// TwinCAT 3 PLC project MainPlc
// ProgramVersion: 3.1.4026.24
// libraries:
//   Tc2_MC2, * (Beckhoff Automation GmbH)
//   Tc2_Standard, * (Beckhoff Automation GmbH)
//   Tc2_System, * (Beckhoff Automation GmbH)
// project tree:
//   DUTs/ ST_AxisData.TcDUT (not stored)
//   GVLs/ GVL_Axis.TcGVL (not stored), GVL_CONSTANT.TcGVL, GVL_PY.TcGVL (not stored)
//   / PlcTask.TcTTO
//   POUs/Axis/ FB_AxisCtrl.TcPOU (not stored), PRG_Enable.TcPOU (not stored), PRG_SineWave.TcPOU (not stored), PRG_Square.TcPOU (not stored)
//   POUs/ MAIN.TcPOU (not stored)
// real-time tasks:
//   TASK PlcTask: cycle T#1ms, priority 20, ADS port 350
// motion (NC):
//   TASK NC-Task 1 SAF: cycle T#1ms, priority 4, ADS port 501
//   TASK NC-Task 1 SVB: cycle T#1ms, priority 8, ADS port 511
//   AXIS Axis 1 (id 1)
//     OtherSettings: AllowMotionCmdToSlave=true
//     encoder EncType=1
//       TimeComp: TimeCompMode=1, EncDelayCycles=4
//     drive DrvType=5
//       Analog: TorqueSetpointScale=10, ScaleFactorActTorque=0.1
//       TimeComp: TimeCompMode=1, TaskDelayCycles=1
//     controller CtrType=1
//       CtrPara: PriorControlFactor=1
//         Observer: BandWidth=20
//   AXIS Axis 2 (id 2)
//     OtherSettings: AllowMotionCmdToSlave=true
//     encoder EncType=1
//     drive DrvType=5
//       Analog: TorqueSetpointScale=10, ScaleFactorActTorque=0.1
//       TimeComp: TaskDelayCycles=1
//     controller CtrType=1
//       CtrPara: PriorControlFactor=1
//         Observer: BandWidth=20
//   AXIS Axis 3 (id 3)
//     OtherSettings: AllowMotionCmdToSlave=true
//     encoder EncType=1
//     drive DrvType=5
//       Analog: TorqueSetpointScale=10, ScaleFactorActTorque=0.1
//       TimeComp: TaskDelayCycles=1
//     controller CtrType=1
//       CtrPara: PriorControlFactor=1
//         Observer: BandWidth=20
//   AXIS Axis 4 (id 4)
//     OtherSettings: AllowMotionCmdToSlave=true
//     encoder EncType=1
//     drive DrvType=5
//       Analog: TorqueSetpointScale=10, ScaleFactorActTorque=0.1
//       TimeComp: TaskDelayCycles=1
//     controller CtrType=1
//       CtrPara: PriorControlFactor=1
//         Observer: BandWidth=20
//   AXIS Axis 5 (id 5)
//     OtherSettings: AllowMotionCmdToSlave=true
//     encoder EncType=1
//     drive DrvType=5
//       Analog: TorqueSetpointScale=10, ScaleFactorActTorque=0.1
//       TimeComp: TaskDelayCycles=1
//     controller CtrType=1
//       CtrPara: PriorControlFactor=1
//         Observer: BandWidth=20
//   AXIS Axis 6 (id 6)
//     OtherSettings: AllowMotionCmdToSlave=true
//     encoder EncType=1
//     drive DrvType=5
//       Analog: TorqueSetpointScale=10, ScaleFactorActTorque=0.1
//       TimeComp: TaskDelayCycles=1
//     controller CtrType=1
//       CtrPara: PriorControlFactor=1
//         Observer: BandWidth=20
//   AXIS Axis 7 (id 7)
//     OtherSettings: AllowMotionCmdToSlave=true
//     encoder EncType=1
//     drive DrvType=5
//       Analog: TorqueSetpointScale=10, ScaleFactorActTorque=0.1
//       TimeComp: TaskDelayCycles=1
//     controller CtrType=1
//       CtrPara: PriorControlFactor=1
//         Observer: BandWidth=20
//   AXIS Axis 8 (id 8)
//     OtherSettings: AllowMotionCmdToSlave=true
//     encoder EncType=1
//     drive DrvType=5
//       Analog: TorqueSetpointScale=10, ScaleFactorActTorque=0.1
//       TimeComp: TaskDelayCycles=1
//     controller CtrType=1
//       CtrPara: PriorControlFactor=1
//         Observer: BandWidth=20
//   AXIS Axis 9 (id 9)
//     OtherSettings: AllowMotionCmdToSlave=true
//     encoder EncType=1
//     drive DrvType=5
//       Analog: TorqueSetpointScale=10, ScaleFactorActTorque=0.1
//       TimeComp: TaskDelayCycles=1
//     controller CtrType=1
//       CtrPara: PriorControlFactor=1
//         Observer: BandWidth=20
//   AXIS Axis 10 (id 10)
//     OtherSettings: AllowMotionCmdToSlave=true
//     encoder EncType=1
//     drive DrvType=5
//       Analog: TorqueSetpointScale=10, ScaleFactorActTorque=0.1
//       TimeComp: TaskDelayCycles=1
//     controller CtrType=1
//       CtrPara: PriorControlFactor=1
//         Observer: BandWidth=20
//   AXIS Axis 11 (id 11)
//     OtherSettings: AllowMotionCmdToSlave=true
//     encoder EncType=1
//     drive DrvType=5
//       Analog: TorqueSetpointScale=10, ScaleFactorActTorque=0.1
//       TimeComp: TaskDelayCycles=1
//     controller CtrType=1
//       CtrPara: PriorControlFactor=1
//         Observer: BandWidth=20
//   AXIS Axis 12 (id 12)
//     OtherSettings: AllowMotionCmdToSlave=true
//     encoder EncType=1
//     drive DrvType=5
//       Analog: TorqueSetpointScale=10, ScaleFactorActTorque=0.1
//       TimeComp: TaskDelayCycles=1
//     controller CtrType=1
//       CtrPara: PriorControlFactor=1
//         Observer: BandWidth=20
//   AXIS Axis 13 (id 13)
//     OtherSettings: AllowMotionCmdToSlave=true
//     encoder EncType=1
//     drive DrvType=5
//       Analog: TorqueSetpointScale=10, ScaleFactorActTorque=0.1
//       TimeComp: TaskDelayCycles=1
//     controller CtrType=1
//       CtrPara: PriorControlFactor=1
//         Observer: BandWidth=20
//   AXIS Axis 14 (id 14)
//     OtherSettings: AllowMotionCmdToSlave=true
//     encoder EncType=1
//     drive DrvType=5
//       Analog: TorqueSetpointScale=10, ScaleFactorActTorque=0.1
//       TimeComp: TaskDelayCycles=1
//     controller CtrType=1
//       CtrPara: PriorControlFactor=1
//         Observer: BandWidth=20
//   AXIS Axis 15 (id 15)
//     OtherSettings: AllowMotionCmdToSlave=true
//     encoder EncType=1
//     drive DrvType=5
//       Analog: TorqueSetpointScale=10, ScaleFactorActTorque=0.1
//       TimeComp: TaskDelayCycles=1
//     controller CtrType=1
//       CtrPara: PriorControlFactor=1
//         Observer: BandWidth=20
//   AXIS Axis 16 (id 16)
//     OtherSettings: AllowMotionCmdToSlave=true
//     encoder EncType=1
//     drive DrvType=5
//       Analog: TorqueSetpointScale=10, ScaleFactorActTorque=0.1
//       TimeComp: TaskDelayCycles=1
//     controller CtrType=1
//       CtrPara: PriorControlFactor=1
//         Observer: BandWidth=20
//   AXIS Axis 17 (id 17)
//     OtherSettings: AllowMotionCmdToSlave=true
//     encoder EncType=1
//     drive DrvType=5
//       Analog: TorqueSetpointScale=10, ScaleFactorActTorque=0.1
//       TimeComp: TaskDelayCycles=1
//     controller CtrType=1
//       CtrPara: PriorControlFactor=1
//         Observer: BandWidth=20
//   AXIS Axis 18 (id 18)
//     OtherSettings: AllowMotionCmdToSlave=true
//     encoder EncType=1
//     drive DrvType=5
//       Analog: TorqueSetpointScale=10, ScaleFactorActTorque=0.1
//       TimeComp: TaskDelayCycles=1
//     controller CtrType=1
//       CtrPara: PriorControlFactor=1
//         Observer: BandWidth=20
//   AXIS Axis 19 (id 19)
//     OtherSettings: AllowMotionCmdToSlave=true
//     encoder EncType=1
//     drive DrvType=5
//       Analog: TorqueSetpointScale=10, ScaleFactorActTorque=0.1
//       TimeComp: TaskDelayCycles=1
//     controller CtrType=1
//       CtrPara: PriorControlFactor=1
//         Observer: BandWidth=20
//   AXIS Axis 20 (id 20)
//     OtherSettings: AllowMotionCmdToSlave=true
//     encoder EncType=1
//     drive DrvType=5
//       Analog: TorqueSetpointScale=10, ScaleFactorActTorque=0.1
//       TimeComp: TaskDelayCycles=1
//     controller CtrType=1
//       CtrPara: PriorControlFactor=1
//         Observer: BandWidth=20
//   AXIS Axis 21 (id 21)
//     OtherSettings: AllowMotionCmdToSlave=true
//     encoder EncType=1
//     drive DrvType=5
//       Analog: TorqueSetpointScale=10, ScaleFactorActTorque=0.1
//       TimeComp: TaskDelayCycles=1
//     controller CtrType=1
//       CtrPara: PriorControlFactor=1
//         Observer: BandWidth=20
//   AXIS Axis 22 (id 22)
//     OtherSettings: AllowMotionCmdToSlave=true
//     encoder EncType=1
//     drive DrvType=5
//       Analog: TorqueSetpointScale=10, ScaleFactorActTorque=0.1
//       TimeComp: TaskDelayCycles=1
//     controller CtrType=1
//       CtrPara: PriorControlFactor=1
//         Observer: BandWidth=20
//   AXIS Axis 23 (id 23)
//     OtherSettings: AllowMotionCmdToSlave=true
//     encoder EncType=1
//     drive DrvType=5
//       Analog: TorqueSetpointScale=10, ScaleFactorActTorque=0.1
//       TimeComp: TaskDelayCycles=1
//     controller CtrType=1
//       CtrPara: PriorControlFactor=1
//         Observer: BandWidth=20
//   AXIS Axis 24 (id 24)
//     OtherSettings: AllowMotionCmdToSlave=true
//     encoder EncType=1
//     drive DrvType=5
//       Analog: TorqueSetpointScale=10, ScaleFactorActTorque=0.1
//       TimeComp: TaskDelayCycles=1
//     controller CtrType=1
//       CtrPara: PriorControlFactor=1
//         Observer: BandWidth=20
//   AXIS Axis 25 (id 25)
//     OtherSettings: AllowMotionCmdToSlave=true
//     encoder EncType=1
//     drive DrvType=5
//       Analog: TorqueSetpointScale=10, ScaleFactorActTorque=0.1
//       TimeComp: TaskDelayCycles=1
//     controller CtrType=1
//       CtrPara: PriorControlFactor=1
//         Observer: BandWidth=20
//   AXIS Axis 26 (id 26)
//     OtherSettings: AllowMotionCmdToSlave=true
//     encoder EncType=1
//     drive DrvType=5
//       Analog: TorqueSetpointScale=10, ScaleFactorActTorque=0.1
//       TimeComp: TaskDelayCycles=1
//     controller CtrType=1
//       CtrPara: PriorControlFactor=1
//         Observer: BandWidth=20
//   AXIS Axis 27 (id 27)
//     OtherSettings: AllowMotionCmdToSlave=true
//     encoder EncType=1
//     drive DrvType=5
//       Analog: TorqueSetpointScale=10, ScaleFactorActTorque=0.1
//       TimeComp: TaskDelayCycles=1
//     controller CtrType=1
//       CtrPara: PriorControlFactor=1
//         Observer: BandWidth=20
//   AXIS Axis 28 (id 28)
//     OtherSettings: AllowMotionCmdToSlave=true
//     encoder EncType=1
//     drive DrvType=5
//       Analog: TorqueSetpointScale=10, ScaleFactorActTorque=0.1
//       TimeComp: TaskDelayCycles=1
//     controller CtrType=1
//       CtrPara: PriorControlFactor=1
//         Observer: BandWidth=20
//   AXIS Axis 29 (id 29)
//     OtherSettings: AllowMotionCmdToSlave=true
//     encoder EncType=1
//     drive DrvType=5
//       Analog: TorqueSetpointScale=10, ScaleFactorActTorque=0.1
//       TimeComp: TaskDelayCycles=1
//     controller CtrType=1
//       CtrPara: PriorControlFactor=1
//         Observer: BandWidth=20
//   AXIS Axis 30 (id 30)
//     OtherSettings: AllowMotionCmdToSlave=true
//     encoder EncType=1
//     drive DrvType=5
//       Analog: TorqueSetpointScale=10, ScaleFactorActTorque=0.1
//       TimeComp: TaskDelayCycles=1
//     controller CtrType=1
//       CtrPara: PriorControlFactor=1
//         Observer: BandWidth=20
//   AXIS Axis 31 (id 31)
//     OtherSettings: AllowMotionCmdToSlave=true
//     encoder EncType=1
//     drive DrvType=5
//       Analog: TorqueSetpointScale=10, ScaleFactorActTorque=0.1
//       TimeComp: TaskDelayCycles=1
//     controller CtrType=1
//       CtrPara: PriorControlFactor=1
//         Observer: BandWidth=20
//   AXIS Axis 32 (id 32)
//     OtherSettings: AllowMotionCmdToSlave=true
//     encoder EncType=1
//     drive DrvType=5
//       Analog: TorqueSetpointScale=10, ScaleFactorActTorque=0.1
//       TimeComp: TaskDelayCycles=1
//     controller CtrType=1
//       CtrPara: PriorControlFactor=1
//         Observer: BandWidth=20
//   AXIS Axis 33 (id 33)
//     OtherSettings: AllowMotionCmdToSlave=true
//     encoder EncType=1
//     drive DrvType=5
//       Analog: TorqueSetpointScale=10, ScaleFactorActTorque=0.1
//       TimeComp: TaskDelayCycles=1
//     controller CtrType=1
//       CtrPara: PriorControlFactor=1
//         Observer: BandWidth=20
//   AXIS Axis 34 (id 34)
//     OtherSettings: AllowMotionCmdToSlave=true
//     encoder EncType=1
//     drive DrvType=5
//       Analog: TorqueSetpointScale=10, ScaleFactorActTorque=0.1
//       TimeComp: TaskDelayCycles=1
//     controller CtrType=1
//       CtrPara: PriorControlFactor=1
//         Observer: BandWidth=20
//   AXIS Axis 35 (id 35)
//     OtherSettings: AllowMotionCmdToSlave=true
//     encoder EncType=1
//     drive DrvType=5
//       Analog: TorqueSetpointScale=10, ScaleFactorActTorque=0.1
//       TimeComp: TaskDelayCycles=1
//     controller CtrType=1
//       CtrPara: PriorControlFactor=1
//         Observer: BandWidth=20
//   AXIS Axis 36 (id 36)
//     OtherSettings: AllowMotionCmdToSlave=true
//     encoder EncType=1
//     drive DrvType=5
//       Analog: TorqueSetpointScale=10, ScaleFactorActTorque=0.1
//       TimeComp: TaskDelayCycles=1
//     controller CtrType=1
//       CtrPara: PriorControlFactor=1
//         Observer: BandWidth=20
// variable links:
//   MainPlc/MainPlc Instance <-> NC-Task 1 SAF/Axes/Axis 1
//     PlcTask Inputs/GVL_Axis.stAxes[1].NcToPlc <-> Outputs/ToPlc
//     PlcTask Outputs/GVL_Axis.stAxes[1].PlcToNc <-> Inputs/FromPlc
//   MainPlc/MainPlc Instance <-> NC-Task 1 SAF/Axes/Axis 10
//     PlcTask Inputs/GVL_Axis.stAxes[10].NcToPlc <-> Outputs/ToPlc
//     PlcTask Outputs/GVL_Axis.stAxes[10].PlcToNc <-> Inputs/FromPlc
//   MainPlc/MainPlc Instance <-> NC-Task 1 SAF/Axes/Axis 11
//     PlcTask Inputs/GVL_Axis.stAxes[11].NcToPlc <-> Outputs/ToPlc
//     PlcTask Outputs/GVL_Axis.stAxes[11].PlcToNc <-> Inputs/FromPlc
//   MainPlc/MainPlc Instance <-> NC-Task 1 SAF/Axes/Axis 12
//     PlcTask Inputs/GVL_Axis.stAxes[12].NcToPlc <-> Outputs/ToPlc
//     PlcTask Outputs/GVL_Axis.stAxes[12].PlcToNc <-> Inputs/FromPlc
//   MainPlc/MainPlc Instance <-> NC-Task 1 SAF/Axes/Axis 13
//     PlcTask Inputs/GVL_Axis.stAxes[13].NcToPlc <-> Outputs/ToPlc
//     PlcTask Outputs/GVL_Axis.stAxes[13].PlcToNc <-> Inputs/FromPlc
//   MainPlc/MainPlc Instance <-> NC-Task 1 SAF/Axes/Axis 14
//     PlcTask Inputs/GVL_Axis.stAxes[14].NcToPlc <-> Outputs/ToPlc
//     PlcTask Outputs/GVL_Axis.stAxes[14].PlcToNc <-> Inputs/FromPlc
//   MainPlc/MainPlc Instance <-> NC-Task 1 SAF/Axes/Axis 15
//     PlcTask Inputs/GVL_Axis.stAxes[15].NcToPlc <-> Outputs/ToPlc
//     PlcTask Outputs/GVL_Axis.stAxes[15].PlcToNc <-> Inputs/FromPlc
//   MainPlc/MainPlc Instance <-> NC-Task 1 SAF/Axes/Axis 16
//     PlcTask Inputs/GVL_Axis.stAxes[16].NcToPlc <-> Outputs/ToPlc
//     PlcTask Outputs/GVL_Axis.stAxes[16].PlcToNc <-> Inputs/FromPlc
//   MainPlc/MainPlc Instance <-> NC-Task 1 SAF/Axes/Axis 17
//     PlcTask Inputs/GVL_Axis.stAxes[17].NcToPlc <-> Outputs/ToPlc
//     PlcTask Outputs/GVL_Axis.stAxes[17].PlcToNc <-> Inputs/FromPlc
//   MainPlc/MainPlc Instance <-> NC-Task 1 SAF/Axes/Axis 18
//     PlcTask Inputs/GVL_Axis.stAxes[18].NcToPlc <-> Outputs/ToPlc
//     PlcTask Outputs/GVL_Axis.stAxes[18].PlcToNc <-> Inputs/FromPlc
//   MainPlc/MainPlc Instance <-> NC-Task 1 SAF/Axes/Axis 19
//     PlcTask Inputs/GVL_Axis.stAxes[19].NcToPlc <-> Outputs/ToPlc
//     PlcTask Outputs/GVL_Axis.stAxes[19].PlcToNc <-> Inputs/FromPlc
//   MainPlc/MainPlc Instance <-> NC-Task 1 SAF/Axes/Axis 2
//     PlcTask Inputs/GVL_Axis.stAxes[2].NcToPlc <-> Outputs/ToPlc
//     PlcTask Outputs/GVL_Axis.stAxes[2].PlcToNc <-> Inputs/FromPlc
//   MainPlc/MainPlc Instance <-> NC-Task 1 SAF/Axes/Axis 20
//     PlcTask Inputs/GVL_Axis.stAxes[20].NcToPlc <-> Outputs/ToPlc
//     PlcTask Outputs/GVL_Axis.stAxes[20].PlcToNc <-> Inputs/FromPlc
//   MainPlc/MainPlc Instance <-> NC-Task 1 SAF/Axes/Axis 21
//     PlcTask Inputs/GVL_Axis.stAxes[21].NcToPlc <-> Outputs/ToPlc
//     PlcTask Outputs/GVL_Axis.stAxes[21].PlcToNc <-> Inputs/FromPlc
//   MainPlc/MainPlc Instance <-> NC-Task 1 SAF/Axes/Axis 22
//     PlcTask Inputs/GVL_Axis.stAxes[22].NcToPlc <-> Outputs/ToPlc
//     PlcTask Outputs/GVL_Axis.stAxes[22].PlcToNc <-> Inputs/FromPlc
//   MainPlc/MainPlc Instance <-> NC-Task 1 SAF/Axes/Axis 23
//     PlcTask Inputs/GVL_Axis.stAxes[23].NcToPlc <-> Outputs/ToPlc
//     PlcTask Outputs/GVL_Axis.stAxes[23].PlcToNc <-> Inputs/FromPlc
//   MainPlc/MainPlc Instance <-> NC-Task 1 SAF/Axes/Axis 24
//     PlcTask Inputs/GVL_Axis.stAxes[24].NcToPlc <-> Outputs/ToPlc
//     PlcTask Outputs/GVL_Axis.stAxes[24].PlcToNc <-> Inputs/FromPlc
//   MainPlc/MainPlc Instance <-> NC-Task 1 SAF/Axes/Axis 25
//     PlcTask Inputs/GVL_Axis.stAxes[25].NcToPlc <-> Outputs/ToPlc
//     PlcTask Outputs/GVL_Axis.stAxes[25].PlcToNc <-> Inputs/FromPlc
//   MainPlc/MainPlc Instance <-> NC-Task 1 SAF/Axes/Axis 26
//     PlcTask Inputs/GVL_Axis.stAxes[26].NcToPlc <-> Outputs/ToPlc
//     PlcTask Outputs/GVL_Axis.stAxes[26].PlcToNc <-> Inputs/FromPlc
//   MainPlc/MainPlc Instance <-> NC-Task 1 SAF/Axes/Axis 27
//     PlcTask Inputs/GVL_Axis.stAxes[27].NcToPlc <-> Outputs/ToPlc
//     PlcTask Outputs/GVL_Axis.stAxes[27].PlcToNc <-> Inputs/FromPlc
//   MainPlc/MainPlc Instance <-> NC-Task 1 SAF/Axes/Axis 28
//     PlcTask Inputs/GVL_Axis.stAxes[28].NcToPlc <-> Outputs/ToPlc
//     PlcTask Outputs/GVL_Axis.stAxes[28].PlcToNc <-> Inputs/FromPlc
//   MainPlc/MainPlc Instance <-> NC-Task 1 SAF/Axes/Axis 29
//     PlcTask Inputs/GVL_Axis.stAxes[29].NcToPlc <-> Outputs/ToPlc
//     PlcTask Outputs/GVL_Axis.stAxes[29].PlcToNc <-> Inputs/FromPlc
//   MainPlc/MainPlc Instance <-> NC-Task 1 SAF/Axes/Axis 3
//     PlcTask Inputs/GVL_Axis.stAxes[3].NcToPlc <-> Outputs/ToPlc
//     PlcTask Outputs/GVL_Axis.stAxes[3].PlcToNc <-> Inputs/FromPlc
//   MainPlc/MainPlc Instance <-> NC-Task 1 SAF/Axes/Axis 30
//     PlcTask Inputs/GVL_Axis.stAxes[30].NcToPlc <-> Outputs/ToPlc
//     PlcTask Outputs/GVL_Axis.stAxes[30].PlcToNc <-> Inputs/FromPlc
//   MainPlc/MainPlc Instance <-> NC-Task 1 SAF/Axes/Axis 31
//     PlcTask Inputs/GVL_Axis.stAxes[31].NcToPlc <-> Outputs/ToPlc
//     PlcTask Outputs/GVL_Axis.stAxes[31].PlcToNc <-> Inputs/FromPlc
//   MainPlc/MainPlc Instance <-> NC-Task 1 SAF/Axes/Axis 32
//     PlcTask Inputs/GVL_Axis.stAxes[32].NcToPlc <-> Outputs/ToPlc
//     PlcTask Outputs/GVL_Axis.stAxes[32].PlcToNc <-> Inputs/FromPlc
//   MainPlc/MainPlc Instance <-> NC-Task 1 SAF/Axes/Axis 33
//     PlcTask Inputs/GVL_Axis.stAxes[33].NcToPlc <-> Outputs/ToPlc
//     PlcTask Outputs/GVL_Axis.stAxes[33].PlcToNc <-> Inputs/FromPlc
//   MainPlc/MainPlc Instance <-> NC-Task 1 SAF/Axes/Axis 34
//     PlcTask Inputs/GVL_Axis.stAxes[34].NcToPlc <-> Outputs/ToPlc
//     PlcTask Outputs/GVL_Axis.stAxes[34].PlcToNc <-> Inputs/FromPlc
//   MainPlc/MainPlc Instance <-> NC-Task 1 SAF/Axes/Axis 35
//     PlcTask Inputs/GVL_Axis.stAxes[35].NcToPlc <-> Outputs/ToPlc
//     PlcTask Outputs/GVL_Axis.stAxes[35].PlcToNc <-> Inputs/FromPlc
//   MainPlc/MainPlc Instance <-> NC-Task 1 SAF/Axes/Axis 36
//     PlcTask Inputs/GVL_Axis.stAxes[36].NcToPlc <-> Outputs/ToPlc
//     PlcTask Outputs/GVL_Axis.stAxes[36].PlcToNc <-> Inputs/FromPlc
//   MainPlc/MainPlc Instance <-> NC-Task 1 SAF/Axes/Axis 4
//     PlcTask Inputs/GVL_Axis.stAxes[4].NcToPlc <-> Outputs/ToPlc
//     PlcTask Outputs/GVL_Axis.stAxes[4].PlcToNc <-> Inputs/FromPlc
//   MainPlc/MainPlc Instance <-> NC-Task 1 SAF/Axes/Axis 5
//     PlcTask Inputs/GVL_Axis.stAxes[5].NcToPlc <-> Outputs/ToPlc
//     PlcTask Outputs/GVL_Axis.stAxes[5].PlcToNc <-> Inputs/FromPlc
//   MainPlc/MainPlc Instance <-> NC-Task 1 SAF/Axes/Axis 6
//     PlcTask Inputs/GVL_Axis.stAxes[6].NcToPlc <-> Outputs/ToPlc
//     PlcTask Outputs/GVL_Axis.stAxes[6].PlcToNc <-> Inputs/FromPlc
//   MainPlc/MainPlc Instance <-> NC-Task 1 SAF/Axes/Axis 7
//     PlcTask Inputs/GVL_Axis.stAxes[7].NcToPlc <-> Outputs/ToPlc
//     PlcTask Outputs/GVL_Axis.stAxes[7].PlcToNc <-> Inputs/FromPlc
//   MainPlc/MainPlc Instance <-> NC-Task 1 SAF/Axes/Axis 8
//     PlcTask Inputs/GVL_Axis.stAxes[8].NcToPlc <-> Outputs/ToPlc
//     PlcTask Outputs/GVL_Axis.stAxes[8].PlcToNc <-> Inputs/FromPlc
//   MainPlc/MainPlc Instance <-> NC-Task 1 SAF/Axes/Axis 9
//     PlcTask Inputs/GVL_Axis.stAxes[9].NcToPlc <-> Outputs/ToPlc
//     PlcTask Outputs/GVL_Axis.stAxes[9].PlcToNc <-> Inputs/FromPlc

CONFIGURATION MainPlc
    RESOURCE PLC ON TwinCAT3
        TASK PlcTask(INTERVAL := T#1ms, PRIORITY := 20);
        PROGRAM MAIN WITH PlcTask : MAIN;
    END_RESOURCE
END_CONFIGURATION

// ---- GVLs/GVL_CONSTANT.TcGVL
VAR_GLOBAL CONSTANT
	// Set this to ANY arbitrary integer. The entire PLC system scales to it automatically.
	MAX_AXES 	: INT 	:= 36; 
END_VAR
